Fanuc KAREL source: kb00009.compact.KL

PROGRAM KB00009
%STACKSIZE=65535
%PRIORITY=65535
%NOLOCKGROUP
VAR
P1 : REAL
P2 : REAL
RESULT : REAL
BEGIN
P1=1.0
P2=1.0
RESULT=ATAN2(P1,P2)
END KB00009
